// TIA Portal V19 export
FUNCTION "POPUP" : Void   // FC6, LAD
{ S7_Optimized_Access := 'TRUE' }
// stored: SetENOAutomatically false
   VAR_TEMP   // added for the SCL form of the ladder/FBD networks
      _w1 : Bool;
      _w2 : Bool;
   END_VAR
BEGIN

REGION Network 1: RINSE-1_START
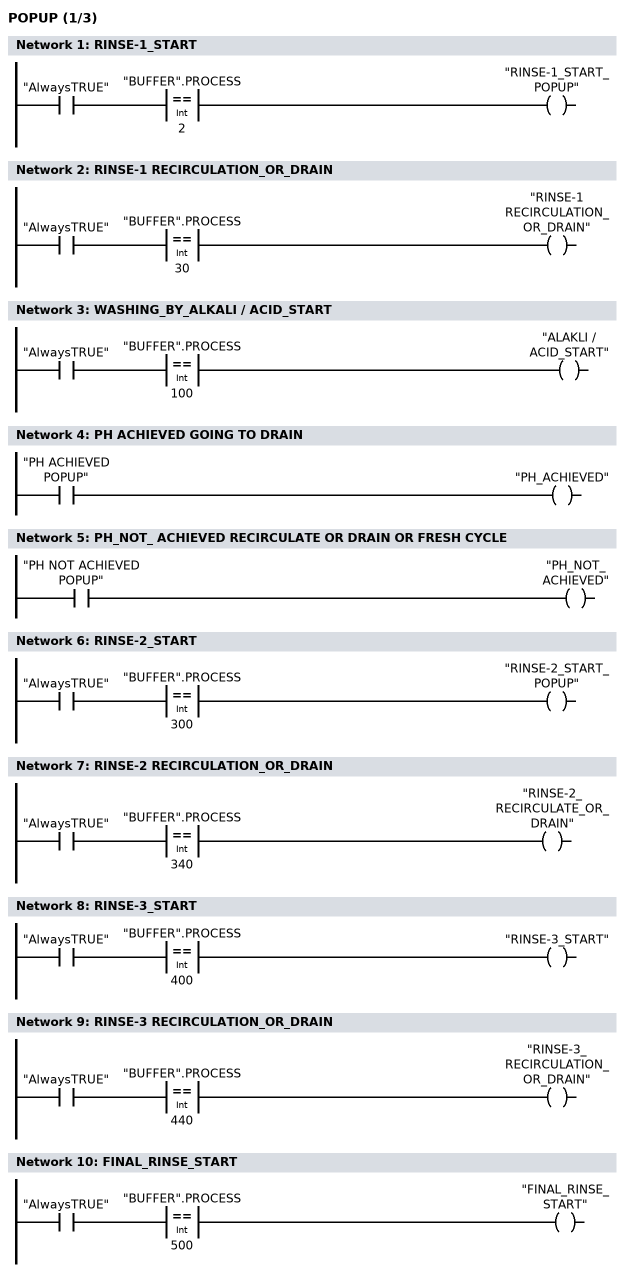
   RUNG wire#powerrail
      Contact( "AlwaysTRUE" )
      { S7_Templates := "SrcType := Int" } EQ_Contact(in1 := "BUFFER".PROCESS, in2 := 2)
      Coil( "RINSE-1_START_POPUP" )
   END_RUNG
   // the same network as SCL:
   "RINSE-1_START_POPUP" := "AlwaysTRUE" AND ("BUFFER".PROCESS = 2);
END_REGION

REGION Network 2: RINSE-1 RECIRCULATION_OR_DRAIN
   RUNG wire#powerrail
      Contact( "AlwaysTRUE" )
      { S7_Templates := "SrcType := Int" } EQ_Contact(in1 := "BUFFER".PROCESS, in2 := 30)
      Coil( "RINSE-1 RECIRCULATION_OR_DRAIN" )
   END_RUNG
   // the same network as SCL:
   "RINSE-1 RECIRCULATION_OR_DRAIN" := "AlwaysTRUE" AND ("BUFFER".PROCESS = 30);
END_REGION

REGION Network 3: WASHING_BY_ALKALI / ACID_START
   RUNG wire#powerrail
      Contact( "AlwaysTRUE" )
      { S7_Templates := "SrcType := Int" } EQ_Contact(in1 := "BUFFER".PROCESS, in2 := 100)
      Coil( "ALAKLI / ACID_START" )
   END_RUNG
   // the same network as SCL:
   "ALAKLI / ACID_START" := "AlwaysTRUE" AND ("BUFFER".PROCESS = 100);
END_REGION

REGION Network 4: PH ACHIEVED GOING TO DRAIN
   RUNG wire#powerrail
      Contact( "PH ACHIEVED POPUP" )
      Coil( "PH_ACHIEVED" )
   END_RUNG
   // the same network as SCL:
   "PH_ACHIEVED" := "PH ACHIEVED POPUP";
END_REGION

REGION Network 5: PH_NOT_ ACHIEVED RECIRCULATE OR DRAIN OR FRESH CYCLE
   RUNG wire#powerrail
      Contact( "PH NOT ACHIEVED POPUP" )
      Coil( "PH_NOT_ACHIEVED" )
   END_RUNG
   // the same network as SCL:
   "PH_NOT_ACHIEVED" := "PH NOT ACHIEVED POPUP";
END_REGION

REGION Network 6: RINSE-2_START
   RUNG wire#powerrail
      Contact( "AlwaysTRUE" )
      { S7_Templates := "SrcType := Int" } EQ_Contact(in1 := "BUFFER".PROCESS, in2 := 300)
      Coil( "RINSE-2_START_POPUP" )
   END_RUNG
   // the same network as SCL:
   "RINSE-2_START_POPUP" := "AlwaysTRUE" AND ("BUFFER".PROCESS = 300);
END_REGION

REGION Network 7: RINSE-2 RECIRCULATION_OR_DRAIN
   RUNG wire#powerrail
      Contact( "AlwaysTRUE" )
      { S7_Templates := "SrcType := Int" } EQ_Contact(in1 := "BUFFER".PROCESS, in2 := 340)
      Coil( "RINSE-2_RECIRCULATE_OR_DRAIN" )
   END_RUNG
   // the same network as SCL:
   "RINSE-2_RECIRCULATE_OR_DRAIN" := "AlwaysTRUE" AND ("BUFFER".PROCESS = 340);
END_REGION

REGION Network 8: RINSE-3_START
   RUNG wire#powerrail
      Contact( "AlwaysTRUE" )
      { S7_Templates := "SrcType := Int" } EQ_Contact(in1 := "BUFFER".PROCESS, in2 := 400)
      Coil( "RINSE-3_START" )
   END_RUNG
   // the same network as SCL:
   "RINSE-3_START" := "AlwaysTRUE" AND ("BUFFER".PROCESS = 400);
END_REGION

REGION Network 9: RINSE-3 RECIRCULATION_OR_DRAIN
   RUNG wire#powerrail
      Contact( "AlwaysTRUE" )
      { S7_Templates := "SrcType := Int" } EQ_Contact(in1 := "BUFFER".PROCESS, in2 := 440)
      Coil( "RINSE-3_RECIRCULATION_OR_DRAIN" )
   END_RUNG
   // the same network as SCL:
   "RINSE-3_RECIRCULATION_OR_DRAIN" := "AlwaysTRUE" AND ("BUFFER".PROCESS = 440);
END_REGION

REGION Network 10: FINAL_RINSE_START
   RUNG wire#powerrail
      Contact( "AlwaysTRUE" )
      { S7_Templates := "SrcType := Int" } EQ_Contact(in1 := "BUFFER".PROCESS, in2 := 500)
      Coil( "FINAL_RINSE_START" )
   END_RUNG
   // the same network as SCL:
   "FINAL_RINSE_START" := "AlwaysTRUE" AND ("BUFFER".PROCESS = 500);
END_REGION

REGION Network 11: CONDUCTIVITY_ACHIEVED
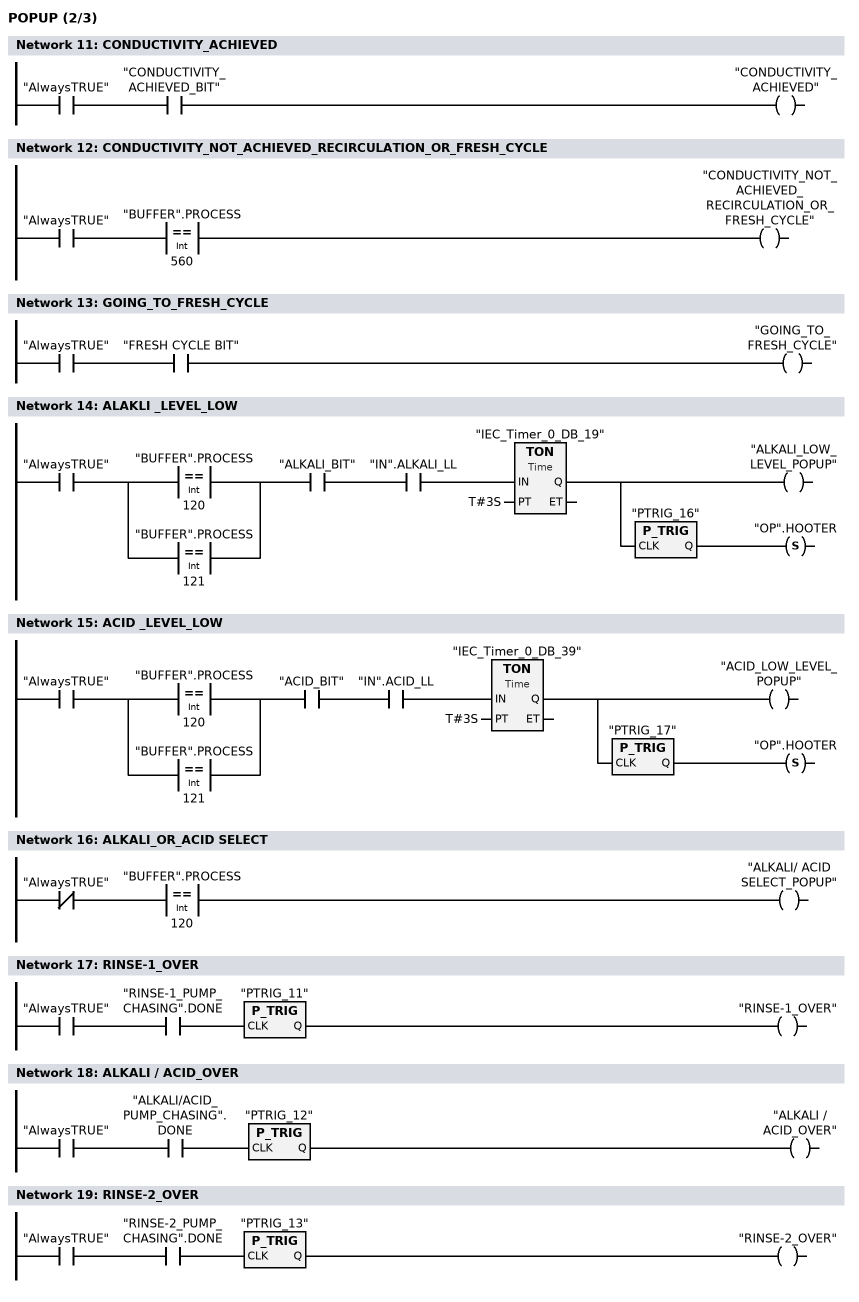
   RUNG wire#powerrail
      Contact( "AlwaysTRUE" )
      Contact( "CONDUCTIVITY_ACHIEVED_BIT" )
      Coil( "CONDUCTIVITY_ACHIEVED" )
   END_RUNG
   // the same network as SCL:
   "CONDUCTIVITY_ACHIEVED" := "AlwaysTRUE" AND "CONDUCTIVITY_ACHIEVED_BIT";
END_REGION

REGION Network 12: CONDUCTIVITY_NOT_ACHIEVED_RECIRCULATION_OR_FRESH_CYCLE
   RUNG wire#powerrail
      Contact( "AlwaysTRUE" )
      { S7_Templates := "SrcType := Int" } EQ_Contact(in1 := "BUFFER".PROCESS, in2 := 560)
      Coil( "CONDUCTIVITY_NOT_ACHIEVED_RECIRCULATION_OR_FRESH_CYCLE" )
   END_RUNG
   // the same network as SCL:
   "CONDUCTIVITY_NOT_ACHIEVED_RECIRCULATION_OR_FRESH_CYCLE" := "AlwaysTRUE" AND ("BUFFER".PROCESS = 560);
END_REGION

REGION Network 13: GOING_TO_FRESH_CYCLE
   RUNG wire#powerrail
      Contact( "AlwaysTRUE" )
      Contact( "FRESH CYCLE BIT" )
      Coil( "GOING_TO_FRESH_CYCLE" )
   END_RUNG
   // the same network as SCL:
   "GOING_TO_FRESH_CYCLE" := "AlwaysTRUE" AND "FRESH CYCLE BIT";
END_REGION

REGION Network 14: ALAKLI _LEVEL_LOW
   RUNG wire#powerrail
      Contact( "AlwaysTRUE" )
      wire#w1
      { S7_Templates := "SrcType := Int" } EQ_Contact(in1 := "BUFFER".PROCESS, in2 := 120)
      wire#w2
      Contact( "ALKALI_BIT" )
      Contact( "IN".ALKALI_LL )
      { S7_Templates := "time_type := Time" } "IEC_Timer_0_DB_19".TON(pt := T#3S, et =>)
      wire#w3
      Coil( "ALKALI_LOW_LEVEL_POPUP" )
   END_RUNG
   RUNG wire#w1
      { S7_Templates := "SrcType := Int" } EQ_Contact(in1 := "BUFFER".PROCESS, in2 := 121)
   END_RUNG wire#w2
   RUNG wire#w3
      P_Trig( "PTRIG_16" )
      S_Coil( "OP".HOOTER )
   END_RUNG
   // the same network as SCL:
   "IEC_Timer_0_DB_19".TON(IN := "AlwaysTRUE" AND (("BUFFER".PROCESS = 120) OR ("BUFFER".PROCESS = 121)) AND "ALKALI_BIT" AND "IN".ALKALI_LL,
                           PT := T#3S);
   "ALKALI_LOW_LEVEL_POPUP" := "IEC_Timer_0_DB_19".Q;
   #_w1 := "IEC_Timer_0_DB_19".Q AND NOT "PTRIG_16";   // rising edge
   "PTRIG_16" := "IEC_Timer_0_DB_19".Q;
   IF #_w1 THEN "OP".HOOTER := TRUE; END_IF;
END_REGION

REGION Network 15: ACID _LEVEL_LOW
   RUNG wire#powerrail
      Contact( "AlwaysTRUE" )
      wire#w1
      { S7_Templates := "SrcType := Int" } EQ_Contact(in1 := "BUFFER".PROCESS, in2 := 120)
      wire#w2
      Contact( "ACID_BIT" )
      Contact( "IN".ACID_LL )
      { S7_Templates := "time_type := Time" } "IEC_Timer_0_DB_39".TON(pt := T#3S, et =>)
      wire#w3
      Coil( "ACID_LOW_LEVEL_POPUP" )
   END_RUNG
   RUNG wire#w1
      { S7_Templates := "SrcType := Int" } EQ_Contact(in1 := "BUFFER".PROCESS, in2 := 121)
   END_RUNG wire#w2
   RUNG wire#w3
      P_Trig( "PTRIG_17" )
      S_Coil( "OP".HOOTER )
   END_RUNG
   // the same network as SCL:
   "IEC_Timer_0_DB_39".TON(IN := "AlwaysTRUE" AND (("BUFFER".PROCESS = 120) OR ("BUFFER".PROCESS = 121)) AND "ACID_BIT" AND "IN".ACID_LL,
                           PT := T#3S);
   "ACID_LOW_LEVEL_POPUP" := "IEC_Timer_0_DB_39".Q;
   #_w1 := "IEC_Timer_0_DB_39".Q AND NOT "PTRIG_17";   // rising edge
   "PTRIG_17" := "IEC_Timer_0_DB_39".Q;
   IF #_w1 THEN "OP".HOOTER := TRUE; END_IF;
END_REGION

REGION Network 16: ALKALI_OR_ACID SELECT
   RUNG wire#powerrail
      I_Contact( "AlwaysTRUE" )
      { S7_Templates := "SrcType := Int" } EQ_Contact(in1 := "BUFFER".PROCESS, in2 := 120)
      Coil( "ALKALI/ ACID SELECT_POPUP" )
   END_RUNG
   // the same network as SCL:
   "ALKALI/ ACID SELECT_POPUP" := NOT "AlwaysTRUE" AND ("BUFFER".PROCESS = 120);
END_REGION

REGION Network 17: RINSE-1_OVER
   RUNG wire#powerrail
      Contact( "AlwaysTRUE" )
      Contact( "RINSE-1_PUMP_CHASING".DONE )
      P_Trig( "PTRIG_11" )
      Coil( "RINSE-1_OVER" )
   END_RUNG
   // the same network as SCL:
   #_w1 := "AlwaysTRUE" AND "RINSE-1_PUMP_CHASING".DONE;
   #_w2 := #_w1 AND NOT "PTRIG_11";   // rising edge
   "PTRIG_11" := #_w1;
   "RINSE-1_OVER" := #_w2;
END_REGION

REGION Network 18: ALKALI / ACID_OVER
   RUNG wire#powerrail
      Contact( "AlwaysTRUE" )
      Contact( "ALKALI/ACID_PUMP_CHASING".DONE )
      P_Trig( "PTRIG_12" )
      Coil( "ALKALI / ACID_OVER" )
   END_RUNG
   // the same network as SCL:
   #_w1 := "AlwaysTRUE" AND "ALKALI/ACID_PUMP_CHASING".DONE;
   #_w2 := #_w1 AND NOT "PTRIG_12";   // rising edge
   "PTRIG_12" := #_w1;
   "ALKALI / ACID_OVER" := #_w2;
END_REGION

REGION Network 19: RINSE-2_OVER
   RUNG wire#powerrail
      Contact( "AlwaysTRUE" )
      Contact( "RINSE-2_PUMP_CHASING".DONE )
      P_Trig( "PTRIG_13" )
      Coil( "RINSE-2_OVER" )
   END_RUNG
   // the same network as SCL:
   #_w1 := "AlwaysTRUE" AND "RINSE-2_PUMP_CHASING".DONE;
   #_w2 := #_w1 AND NOT "PTRIG_13";   // rising edge
   "PTRIG_13" := #_w1;
   "RINSE-2_OVER" := #_w2;
END_REGION

REGION Network 20: FINAL RINSE-1_OVER
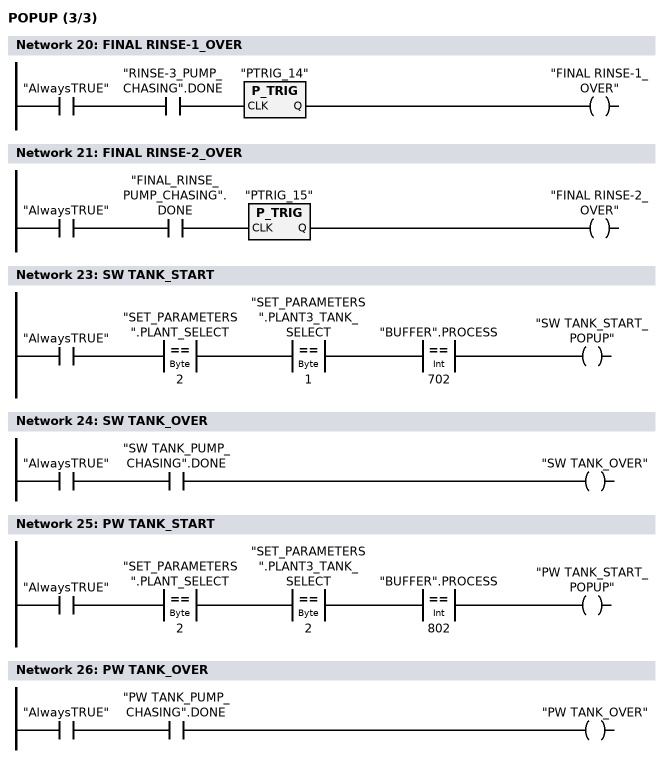
   RUNG wire#powerrail
      Contact( "AlwaysTRUE" )
      Contact( "RINSE-3_PUMP_CHASING".DONE )
      P_Trig( "PTRIG_14" )
      Coil( "FINAL RINSE-1_OVER" )
   END_RUNG
   // the same network as SCL:
   #_w1 := "AlwaysTRUE" AND "RINSE-3_PUMP_CHASING".DONE;
   #_w2 := #_w1 AND NOT "PTRIG_14";   // rising edge
   "PTRIG_14" := #_w1;
   "FINAL RINSE-1_OVER" := #_w2;
END_REGION

REGION Network 21: FINAL RINSE-2_OVER
   RUNG wire#powerrail
      Contact( "AlwaysTRUE" )
      Contact( "FINAL_RINSE_PUMP_CHASING".DONE )
      P_Trig( "PTRIG_15" )
      Coil( "FINAL RINSE-2_OVER" )
   END_RUNG
   // the same network as SCL:
   #_w1 := "AlwaysTRUE" AND "FINAL_RINSE_PUMP_CHASING".DONE;
   #_w2 := #_w1 AND NOT "PTRIG_15";   // rising edge
   "PTRIG_15" := #_w1;
   "FINAL RINSE-2_OVER" := #_w2;
END_REGION

REGION Network 22: ------------NEW LOGIC ADD-----------
END_REGION

REGION Network 23: SW TANK_START
   RUNG wire#powerrail
      Contact( "AlwaysTRUE" )
      { S7_Templates := "SrcType := Byte" } EQ_Contact(in1 := "SET_PARAMETERS".PLANT_SELECT, in2 := 2)
      { S7_Templates := "SrcType := Byte" } EQ_Contact(in1 := "SET_PARAMETERS".PLANT3_TANK_SELECT, in2 := 1)
      { S7_Templates := "SrcType := Int" } EQ_Contact(in1 := "BUFFER".PROCESS, in2 := 702)
      Coil( "SW TANK_START_POPUP" )
   END_RUNG
   // the same network as SCL:
   "SW TANK_START_POPUP" := "AlwaysTRUE" AND ("SET_PARAMETERS".PLANT_SELECT = 2) AND ("SET_PARAMETERS".PLANT3_TANK_SELECT = 1) AND ("BUFFER".PROCESS = 702);
END_REGION

REGION Network 24: SW TANK_OVER
   RUNG wire#powerrail
      Contact( "AlwaysTRUE" )
      Contact( "SW TANK_PUMP_CHASING".DONE )
      Coil( "SW TANK_OVER" )
   END_RUNG
   // the same network as SCL:
   "SW TANK_OVER" := "AlwaysTRUE" AND "SW TANK_PUMP_CHASING".DONE;
END_REGION

REGION Network 25: PW TANK_START
   RUNG wire#powerrail
      Contact( "AlwaysTRUE" )
      { S7_Templates := "SrcType := Byte" } EQ_Contact(in1 := "SET_PARAMETERS".PLANT_SELECT, in2 := 2)
      { S7_Templates := "SrcType := Byte" } EQ_Contact(in1 := "SET_PARAMETERS".PLANT3_TANK_SELECT, in2 := 2)
      { S7_Templates := "SrcType := Int" } EQ_Contact(in1 := "BUFFER".PROCESS, in2 := 802)
      Coil( "PW TANK_START_POPUP" )
   END_RUNG
   // the same network as SCL:
   "PW TANK_START_POPUP" := "AlwaysTRUE" AND ("SET_PARAMETERS".PLANT_SELECT = 2) AND ("SET_PARAMETERS".PLANT3_TANK_SELECT = 2) AND ("BUFFER".PROCESS = 802);
END_REGION

REGION Network 26: PW TANK_OVER
   RUNG wire#powerrail
      Contact( "AlwaysTRUE" )
      Contact( "PW TANK_PUMP_CHASING".DONE )
      Coil( "PW TANK_OVER" )
   END_RUNG
   // the same network as SCL:
   "PW TANK_OVER" := "AlwaysTRUE" AND "PW TANK_PUMP_CHASING".DONE;
END_REGION
END_FUNCTION
